// TwinCAT 3 PLC project PLC_Project
// ProgramVersion: 3.1.4026.19
// CompilerDefines: VISU_USEPROPERTYINFO,VISU_USEWSTRING
// libraries:
//   Tc2_Standard, * (Beckhoff Automation GmbH)
//   Tc2_System, * (Beckhoff Automation GmbH)
//   Tc2_Utilities, * (Beckhoff Automation GmbH)
//   Tc3_EventLogger, * (Beckhoff Automation GmbH)
//   VisuElemEventTable, * (System)
//   VisuSymbols, 4.5.0.0 (System)
// project tree:
//   DUTs/ ST_AlarmEventData_TextList.TcDUT, ST_AlarmEventData_Table.TcDUT
//   FBs/ FB_AlarmEx.TcPOU, FB_Message.TcPOU
//   / GlobalTextList.TcGTLO, PlcTask.TcTTO, Visualization Manager.TcVMO (not stored), VISU_TASK.TcTTO
//   GVLs/ HMI.TcGVL, SYS.TcGVL
//   POUs/ FB_AlarmLogEvent_TextList.TcPOU, FB_AlarmLogEvent_Table.TcPOU, MAIN.TcPOU
//   VISUs/ Alarms.TcVIS, Event_Table.TcVIS, Alarm_Table.TcVIS, Alarm_TextList.TcTLO, stAlarmEventData_TextList.TcTLO
//   VISUs/Frames/ AlarmRow.TcVIS, Alarm_Frame.TcVIS
// real-time tasks:
//   TASK PlcTask: cycle T#10ms, priority 20, ADS port 350
//   TASK VISU_TASK: cycle T#200000us, priority 30, ADS port 351
// I/O:
//   DEVICE Device 1 (EtherCAT) (disabled), AmsNetId 10.0.3.0.2.1
// variable links:
//   PLC_Project/PLC_Project Instance <-> Device 1 (EtherCAT)
//     PlcTask Inputs/MAIN.DevState <-> Inputs/DevState

CONFIGURATION PLC_Project
    RESOURCE PLC ON TwinCAT3
        TASK PlcTask(INTERVAL := T#10ms, PRIORITY := 20);
        TASK VISU_TASK(INTERVAL := T#200000us, PRIORITY := 30);
        PROGRAM MAIN WITH PlcTask : MAIN;
        PROGRAM VisuElems_Visu_Prg WITH VISU_TASK : VisuElems.Visu_Prg;
    END_RESOURCE
END_CONFIGURATION

// ---- DUTs/ST_AlarmEventData_TextList.TcDUT
TYPE ST_AlarmEventData_TextList :
STRUCT
	qActive		: BOOL;
	diEventID	: DINT;
	iClass		: INT; 		//0 = none, 1= Maintenance, 2= Message, 3= Hint, 4= StateInfo, 5= Instruction, 6 = Warning, 7= Alarm, 8= Parameter
	sTime		: STRING;
END_STRUCT
END_TYPE

// ---- DUTs/ST_AlarmEventData_Table.TcDUT
TYPE ST_AlarmEventData_Table :
STRUCT
	qActive		: BOOL;
	diEventID	: DINT;
	iClass		: INT; 		//0 = none, 1= Maintenance, 2= Message, 3= Hint, 4= StateInfo, 5= Instruction, 6 = Warning, 7= Alarm, 8= Parameter
	sTime		: STRING;
	sEvent		: STRING; 	// Event Text
END_STRUCT
END_TYPE

// ---- GVLs/HMI.TcGVL
{attribute 'qualified_only'}
VAR_GLOBAL
astActiveAlarmsList		: ARRAY [0..10] OF ST_AlarmEventData_TextList; // Display list of 10 active alarms, any more than that are just snowballs anyway so why display	
astActiveAlarmsTable	: ARRAY [1..50] OF ST_AlarmEventData_Table; // Display list of 50 active alarms
//Common Controls
	xFaultResetPB			: BOOL; //HMI Fault Reset PB
	xFaultPresent			: BOOL; //HMI Fault Present Indicator
END_VAR

// ---- GVLs/SYS.TcGVL
{attribute 'qualified_only'}
VAR_GLOBAL CONSTANT
iMaxSpeedConstant 		: INT := 60;
END_VAR

{attribute 'qualified_only'}
VAR_GLOBAL RETAIN
	
END_VAR

{attribute 'qualified_only'}
VAR_GLOBAL
	
//Program Declarations
	xFirstScan				: BOOL := TRUE;;
	xFaultPresent			: BOOL;
	ftrigFaultReset			: F_TRIG;
	xFaultReset				: BOOL;

//System Info
	fbGetLocalSystemTIme	: FB_LocalSystemTime;
	sSystemDateTime 		: STRING;
	sSystemTime 			: STRING;
	sSystemDate 			: STRING;
END_VAR

// ---- POUs/MAIN.TcPOU
PROGRAM MAIN
VAR
	DevState AT %I*			: UINT;
	fbReadEvents			: FB_ReadTc3Events; // Required for Event Table Visu Control
	fbMachineAlarm			: ARRAY[0..100] OF FB_AlarmEx;
	fbMachineMessage		: ARRAY[0..100] OF FB_Message;
	TestAlarm				: ARRAY[1..10] OF BOOL;
	TestMessage				: ARRAY[1..10] OF BOOL;
	
	ClearTable				: BOOL;
	VisuSeverity			: ARRAY[0..4] OF STRING := ['Verbose', 'Info', 'Warning', 'Error', 'Critical']; // Used in the Visu Combobox
	Severity				: TcEventSeverity;

	Fault 					: ARRAY [1..100] OF BOOL;
	fbAlarmLogEvent 		: ARRAY [1..100] OF FB_AlarmLogEvent_TextList; //Alarm Logging Event Handler
	fbAlarmLogEventTable	: ARRAY [1..100] OF FB_AlarmLogEvent_Table; //Alarm Logging Event Handler
	iFaultIndex				: INT;
	iAlarmClearIndex		: INT;
	iAlarmActiveIndex		: INT;
	iAlarmActiveIndex2		: INT;
	diAlarmEventLogIndex	: DINT;
END_VAR

//Get Local System Time
	SYS.fbGetLocalSystemTIme( 
		bEnable:= TRUE, 
		dwCycle:= 1);
	//Seperate Date and time
		SYS.sSystemDateTime := SYSTEMTIME_TO_STRING(in:= SYS.fbGetLocalSystemTIme.systemTime);
		SYS.sSystemDate := MID(STR:= SYS.sSystemDateTime, LEN:= 10 , POS:= 1 );
		SYS.sSystemTime := MID(STR:= SYS.sSystemDateTime, LEN:= 8 , POS:= 12 );

// HMI Fault PB Passthrough		
SYS.xFaultReset := HMI.xFaultResetPB;


	
// Twincat Event Logger	
// The function block enables the events of the TwinCAT 3 EventLogger to be displayed in the visualization element event table. 
// FB_ReadTc3Events is contained in the VisuElemEventTable library, which is automatically added to the project when the event table is activated
fbReadEvents(
	bReadEvents := TRUE,										// This input is used to enable the events to be read.
	nLanguageID := 1033,										// Defines which translation of the event text is to be retrieved. 1033 = English
	eDateAndTimeFormat := E_DateAndTimeFormat.en_US,			// Defines the format of the timestamps. E_DateAndTimeFormat
	bClearTable :=	ClearTable,					// The event table is cleared via a positive edge at this input. Alarms that were not acknowledged or reset are not removed from the table.
	eMinSeverity := Severity,									// Only events whose severity is at least as high as the severity specified here are displayed in the event table.
	aEvents => ,												// The function block uses this array to make the evaluated events available. The array can store a maximum of 80 messages. If the number of events is large, older messages are overwritten.
	nNumberOfEvents => ,										// Indicates how many events were triggered.
	bError => ,													// This output is set if an error occurs when polling or processing the events.
	hrErrorCode => );											// Indicates the error code of the error that has occurred.

Tc3_EventLogger();





// Legacy Alarm List
A99_Alarms_TextList();
A99_Alarms_Table();

// First Scan Complete
SYS.xFirstScan := FALSE;

ACTION A99_Alarms_Table:
//System Faults
	//Power Interrupted Fault							
		fbAlarmLogEventTable[1](
							i_diEventID:= 1,							// Must match the AlarmText Index for the message to display
							sEventText := 'Power Interrupt Fault',		// Enter an Event String Here
							i_iClassID:= 7,								// 0 = none, 1= Maintenance, 2= Message, 3= Hint, 4= StateInfo, 5= Instruction, 6 = Warning, 7= Alarm, 8= Paramater		
							bSetEvent := SYS.xFirstScan,				// Event activates on rising edge, clears on falling edge
							bLatchTillAck:= TRUE,						// Option to Latch alarm on even if no longer active, wait till alarm ack to clear
							bAck:= SYS.xFaultReset);					// Acknowledged and clears on rising edge if option LatchTillAck = false
							

		fbAlarmLogEventTable[2](
							i_diEventID:= 2,
							sEventText := 'Test Alarm 1',
							i_iClassID:= 7,
							bSetEvent := TestAlarm[1],
							bLatchTillAck:= TRUE,
							bAck:= SYS.xFaultReset);
							

		fbAlarmLogEventTable[3](
							i_diEventID:= 3,
							sEventText := 'Test Alarm 2',
							i_iClassID:= 2,
							bSetEvent := TestAlarm[2],
							bLatchTillAck:= TRUE,
							bAck:= SYS.xFaultReset);
							
					
		fbAlarmLogEventTable[4](
							i_diEventID:= 4,
							sEventText := 'Test Alarm 3',
							i_iClassID:= 6,
							bSetEvent := TestAlarm[3],
							bLatchTillAck:= TRUE,
							bAck:= SYS.xFaultReset);
							
				
		fbAlarmLogEventTable[5](
							i_diEventID:= 5,
							sEventText := 'Test Alarm 4',
							i_iClassID:= 7,
							bSetEvent := TestAlarm[4],
							bLatchTillAck:= TRUE,
							bAck:= SYS.xFaultReset);


// iClassID : 0 = none, 1= Maintenance, 2= Message, 3= Hint, 4= StateInfo, 5= Instruction, 6 = Warning, 7= Alarm, 8= Paramater	
//Monitor Fault Present
FOR iFaultIndex := 1 TO 100 BY 1 DO
	//System
	IF (iFaultIndex > 0) AND (iFaultIndex < 20) THEN // Look at Alarm Group 1-20
		IF fbAlarmLogEventTable[iFaultIndex].q_xActive AND (fbAlarmLogEventTable[iFaultIndex].i_iClassID = 7) THEN // Only Class 7 Count as Alarms
			SYS.xFaultPresent := TRUE;
		END_IF
	END_IF
	
(*  Some Other Alarm Group
	IF (iFaultIndex >= 20) AND (iFaultIndex < 40) THEN // Subsequent Alarm Group
		IF fbAlarmLogEvent[iFaultIndex].q_xActive AND (fbAlarmLogEvent[iFaultIndex].i_iClassID = 7) THEN
			OtherMachineFaultPreset := TRUE;
		END_IF
	END_IF
*)
END_FOR

// System Fault to HMI Fault Indicator
HMI.xFaultPresent := SYS.xFaultPresent;

IF SYS.xFaultReset THEN
	SYS.xFaultPresent := FALSE;
END_IF

(* Log all Alarms using the fbAlarmLogEvent function block*)
(* Alarm Text is in the Alarm_TextList File*)	

//Clear active alarms list before re-populating to ensure old cleared alarms are not stranded in the list
IF SYS.xFaultReset THEN
	FOR iAlarmClearIndex := 1 TO 50 BY 1 DO //10 possible active Alarms, no more!
		HMI.astActiveAlarmsTable[iAlarmClearIndex].sEvent := '';
		HMI.astActiveAlarmsTable[iAlarmClearIndex].diEventID := 0;
		HMI.astActiveAlarmsTable[iAlarmClearIndex].iClass := 0;
		HMI.astActiveAlarmsTable[iAlarmClearIndex].sTime := '';
	END_FOR;
END_IF
	
//Populate HMI Active Alarms list
	iAlarmActiveIndex2 := 0;  //Initialize before seeing how many active alarms there are.
	FOR diAlarmEventLogIndex := 1 TO 100 BY 1 DO //100 possible defined Alarms, no more!
		IF fbAlarmLogEvent[diAlarmEventLogIndex].q_xActive THEN
			IF iAlarmActiveIndex2 <= 9 THEN //10 max active alarms, no more!
				iAlarmActiveIndex2 := iAlarmActiveIndex2 + 1;
			END_IF
			HMI.astActiveAlarmsTable[iAlarmActiveIndex2].sEvent := fbAlarmLogEventTable[diAlarmEventLogIndex].q_stAlarmEventData.sEvent;
			HMI.astActiveAlarmsTable[iAlarmActiveIndex2].diEventID := fbAlarmLogEventTable[diAlarmEventLogIndex].q_stAlarmEventData.diEventID;
			HMI.astActiveAlarmsTable[iAlarmActiveIndex2].iClass := fbAlarmLogEventTable[diAlarmEventLogIndex].q_stAlarmEventData.iClass;
			IF HMI.astActiveAlarmsTable[iAlarmActiveIndex2].sTime = '' THEN
				HMI.astActiveAlarmsTable[iAlarmActiveIndex2].sTime := SYS.sSystemTime;
			END_IF
		END_IF
	END_FOR;
END_ACTION

ACTION A99_Alarms_TextList:
//System Faults
	//Power Interrupted Fault
		fbAlarmLogEvent[1](i_diEventID:= 1,					// Must match the AlarmText Index for the message to display
							i_iClassID:= 7,					// 0 = none, 1= Maintenance, 2= Message, 3= Hint, 4= StateInfo, 5= Instruction, 6 = Warning, 7= Alarm, 8= Paramater		
							bSetEvent := SYS.xFirstScan,	// Event activates on rising edge, clears on falling edge
							bLatchTillAck:= TRUE,			// Option to Latch alarm on even if no longer active, wait till alarm ack to clear
							bAck:= SYS.xFaultReset);		// Acknowledged and clears on rising edge if option LatchTillAck = false
							

		fbAlarmLogEvent[2](i_diEventID:= 2,
							i_iClassID:= 7,
							bSetEvent := TestAlarm[1],
							bLatchTillAck:= TRUE,
							bAck:= SYS.xFaultReset);
							

		fbAlarmLogEvent[3](i_diEventID:= 3,
							i_iClassID:= 2,
							bSetEvent := TestAlarm[2],
							bLatchTillAck:= TRUE,
							bAck:= SYS.xFaultReset);
							
					
		fbAlarmLogEvent[4](i_diEventID:= 4,
							i_iClassID:= 6,
							bSetEvent := TestAlarm[3],
							bLatchTillAck:= TRUE,
							bAck:= SYS.xFaultReset);
							
				
		fbAlarmLogEvent[5](i_diEventID:= 5,
							i_iClassID:= 7,
							bSetEvent := TestAlarm[4],
							bLatchTillAck:= TRUE,
							bAck:= SYS.xFaultReset);


// iClassID : 0 = none, 1= Maintenance, 2= Message, 3= Hint, 4= StateInfo, 5= Instruction, 6 = Warning, 7= Alarm, 8= Paramater	
//Monitor Fault Present
FOR iFaultIndex := 1 TO 100 BY 1 DO
	//System
	IF (iFaultIndex > 0) AND (iFaultIndex < 20) THEN // Look at Alarm Group 1-20
		IF fbAlarmLogEvent[iFaultIndex].q_xActive AND (fbAlarmLogEvent[iFaultIndex].i_iClassID = 7) THEN // Only Class 7 Count as Alarms
			SYS.xFaultPresent := TRUE;
		END_IF
	END_IF
	
(*  Some Other Alarm Group
	IF (iFaultIndex >= 20) AND (iFaultIndex < 40) THEN // Subsequent Alarm Group
		IF fbAlarmLogEvent[iFaultIndex].q_xActive AND (fbAlarmLogEvent[iFaultIndex].i_iClassID = 7) THEN
			OtherMachineFaultPreset := TRUE;
		END_IF
	END_IF
*)
END_FOR

// System Fault to HMI Fault Indicator
HMI.xFaultPresent := SYS.xFaultPresent;

IF SYS.xFaultReset THEN
	SYS.xFaultPresent := FALSE;
END_IF

(* Log all Alarms using the fbAlarmLogEvent function block*)
(* Alarm Text is in the Alarm_TextList File*)	

//Clear active alarms list before re-populating to ensure old cleared alarms are not stranded in the list
IF SYS.xFaultReset THEN
	FOR iAlarmClearIndex := 0 TO 10 BY 1 DO //10 possible active Alarms, no more!
		HMI.astActiveAlarmsList[iAlarmClearIndex].diEventID := 0;
		HMI.astActiveAlarmsList[iAlarmClearIndex].iClass := 0;
		HMI.astActiveAlarmsList[iAlarmClearIndex].sTime := '';
	END_FOR;
END_IF
	
//Populate HMI Active Alarms list
	iAlarmActiveIndex := 0;  //Initialize before seeing how many active alarms there are.
	FOR diAlarmEventLogIndex := 1 TO 100 BY 1 DO //100 possible defined Alarms, no more!
		IF fbAlarmLogEvent[diAlarmEventLogIndex].q_xActive THEN
			IF iAlarmActiveIndex <= 9 THEN //10 max active alarms, no more!
				iAlarmActiveIndex := iAlarmActiveIndex + 1;
			END_IF
			HMI.astActiveAlarmsList[iAlarmActiveIndex].diEventID := fbAlarmLogEvent[diAlarmEventLogIndex].q_stAlarmEventData.diEventID;
			HMI.astActiveAlarmsList[iAlarmActiveIndex].iClass := fbAlarmLogEvent[diAlarmEventLogIndex].q_stAlarmEventData.iClass;
			IF HMI.astActiveAlarmsList[iAlarmActiveIndex].sTime = '' THEN
				HMI.astActiveAlarmsList[iAlarmActiveIndex].sTime := SYS.sSystemTime;
			END_IF
		END_IF
	END_FOR;
END_ACTION

ACTION TC3_EventLogger:
// Event Classes are created in System -> Type System -> Event Class
// Write Click and Create your new Event Class.

fbMachineMessage[1](
	evtEntry:= TC_EVENTS.Test_EventClass.Test_Message1, 
	bEvt:= TestMessage[1]);
	
fbMachineMessage[2](
	evtEntry:= TC_EVENTS.Test_EventClass.Test_Message2, 
	bEvt:= TestMessage[2]);
	
fbMachineMessage[3](
	evtEntry:= TC_EVENTS.Test_EventClass.Test_Message3, 
	bEvt:= TestMessage[3]);
	
fbMachineMessage[4](
	evtEntry:= TC_EVENTS.Test_EventClass.Test_Message4, 
	bEvt:= TestMessage[4]);
	
fbMachineMessage[5](
	evtEntry:= TC_EVENTS.Test_EventClass.Test_Message5, 
	bEvt:= TestMessage[5]);
	
fbMachineAlarm[1](
	evtEntry:= TC_EVENTS.Test_EventClass.PowerInterrupt, 
	bEvt:= SYS.xFirstScan,
	bConfirm := SYS.xFaultReset); 
	
fbMachineAlarm[2](
	evtEntry:= TC_EVENTS.Test_EventClass.Test_Event1, 
	bEvt:= TestAlarm[1],
	bConfirm := SYS.xFaultReset); 
	
fbMachineAlarm[3](
	evtEntry:= TC_EVENTS.Test_EventClass.Test_Event2, 
	bEvt:= TestAlarm[2],
	bConfirm := SYS.xFaultReset); 
	
fbMachineAlarm[4](
	evtEntry:= TC_EVENTS.Test_EventClass.Test_Event3, 
	bEvt:= TestAlarm[3],
	bConfirm := SYS.xFaultReset); 
	
fbMachineAlarm[5](
	evtEntry:= TC_EVENTS.Test_EventClass.Test_Event4, 
	bEvt:= TestAlarm[4],
	bConfirm := SYS.xFaultReset); 


// Trigger Several Alarms At Once below.
// Change Severity in the Event Class	
	
fbMachineAlarm[6](
	evtEntry:= TC_EVENTS.Events._IECCONF_1, 
	bEvt:= TestAlarm[5],
	bConfirm := SYS.xFaultReset); 
	
fbMachineAlarm[7](
	evtEntry:= TC_EVENTS.Events._IECCONF_2, 
	bEvt:= TestAlarm[5],
	bConfirm := SYS.xFaultReset);
	
fbMachineAlarm[8](
	evtEntry:= TC_EVENTS.Events._IECCONF_3, 
	bEvt:= TestAlarm[5],
	bConfirm := SYS.xFaultReset);
	
fbMachineAlarm[9](
	evtEntry:= TC_EVENTS.Events._IECCONF_4, 
	bEvt:= TestAlarm[5],
	bConfirm := SYS.xFaultReset);
	
fbMachineAlarm[10](
	evtEntry:= TC_EVENTS.Events._IECCONF_5, 
	bEvt:= TestAlarm[5],
	bConfirm := SYS.xFaultReset);
	
fbMachineAlarm[11](
	evtEntry:= TC_EVENTS.Events._IECCONF_6, 
	bEvt:= TestAlarm[5],
	bConfirm := SYS.xFaultReset);
	
fbMachineAlarm[12](
	evtEntry:= TC_EVENTS.Events._IECCONF_7, 
	bEvt:= TestAlarm[5],
	bConfirm := SYS.xFaultReset);
	
fbMachineAlarm[13](
	evtEntry:= TC_EVENTS.Events._IECCONF_8, 
	bEvt:= TestAlarm[5],
	bConfirm := SYS.xFaultReset);
	
fbMachineAlarm[14](
	evtEntry:= TC_EVENTS.Events._IECCONF_9, 
	bEvt:= TestAlarm[5],
	bConfirm := SYS.xFaultReset);
	
fbMachineAlarm[15](
	evtEntry:= TC_EVENTS.Events._IECCONF_10, 
	bEvt:= TestAlarm[5],
	bConfirm := SYS.xFaultReset);
	
fbMachineAlarm[16](
	evtEntry:= TC_EVENTS.Events._IECCONF_11, 
	bEvt:= TestAlarm[5],
	bConfirm := SYS.xFaultReset);
	
fbMachineAlarm[17](
	evtEntry:= TC_EVENTS.Events._IECCONF_12, 
	bEvt:= TestAlarm[5],
	bConfirm := SYS.xFaultReset);
	
fbMachineAlarm[18](
	evtEntry:= TC_EVENTS.Events._IECCONF_13, 
	bEvt:= TestAlarm[5],
	bConfirm := SYS.xFaultReset);
	
fbMachineAlarm[19](
	evtEntry:= TC_EVENTS.Events._IECCONF_14, 
	bEvt:= TestAlarm[5],
	bConfirm := SYS.xFaultReset);
	
fbMachineAlarm[20](
	evtEntry:= TC_EVENTS.Events._IECCONF_15, 
	bEvt:= TestAlarm[5],
	bConfirm := SYS.xFaultReset);
	
fbMachineAlarm[21](
	evtEntry:= TC_EVENTS.Events._IECCONF_16, 
	bEvt:= TestAlarm[5],
	bConfirm := SYS.xFaultReset);
	
fbMachineAlarm[22](
	evtEntry:= TC_EVENTS.Events._IECCONF_17, 
	bEvt:= TestAlarm[5],
	bConfirm := SYS.xFaultReset);
END_ACTION

END_PROGRAM

// ---- FBs/FB_AlarmEx.TcPOU
FUNCTION_BLOCK FB_AlarmEx EXTENDS FB_TcAlarm
VAR_INPUT
	evtEntry	: TcEventEntry;
	bEvt		: BOOL;
	bConfirm	: BOOL;
END_VAR
VAR_OUTPUT
END_VAR
VAR
	SourceInfo	: FB_TcSourceInfo;
	bInit	: BOOL := TRUE;
	bMem	: BOOL;
END_VAR

IF bInit THEN
	SUPER^.CreateEx(evtEntry, (evtentry.eSeverity = TcEventSeverity.Critical) OR (evtentry.eSeverity = TcEventSeverity.Error), 0);
	bInit := FALSE;
END_IF

IF bEvt AND NOT bMem AND SUPER^.eConfirmationState <> TcEventConfirmationState.WaitForConfirmation THEN
	SUPER^.Raise(0);
END_IF

IF bMem AND NOT bEvt THEN
	SUPER^.Clear(0,FALSE);
END_IF

IF bConfirm THEN
	SUPER^.Confirm(0);
END_IF

bMem := bEvt;

END_FUNCTION_BLOCK

// ---- FBs/FB_Message.TcPOU
FUNCTION_BLOCK FB_Message EXTENDS FB_TcMessage
VAR_INPUT
	evtEntry	: TcEventEntry;
	bEvt		: BOOL;
END_VAR
VAR_OUTPUT
	bSent		: BOOL;
END_VAR
VAR
	rtrigSend	: R_TRIG;
	bInit	: BOOL := TRUE;
	bMem	: BOOL;
END_VAR

bSent := FALSE;
IF bInit THEN
	SUPER^.CreateEx(stEventEntry := evtEntry, ipSourceInfo := 0);
	bInit := FALSE;
END_IF

rtrigSend(CLK:= bEvt);
IF rtrigSend.Q THEN
	SUPER^.Send(0);
	bSent := TRUE;
END_IF

END_FUNCTION_BLOCK

// ---- POUs/FB_AlarmLogEvent_TextList.TcPOU
FUNCTION_BLOCK FB_AlarmLogEvent_TextList
VAR_INPUT
	bSetEvent			: BOOL;	//Trigger to activate the Alarm
	i_diEventID			: DINT;
	i_iClassID			: INT;
	bLatchTillAck 		: BOOL; //Latch Alarm active till Acked even if alarm event clears.
	bAck				: BOOL; //Acknowledge the alarm and clear it.
	tsTime				:TIMESTRUCT;
END_VAR
VAR_OUTPUT
	q_stAlarmEventData	: ST_AlarmEventData_TextList;
	q_xActive			: BOOL;
END_VAR
VAR
	fbFormatString		: FB_FormatString;
END_VAR

//Why use a Function Block?
//So we could add a active time/date stamp
//So we could add to a historical alarm area
//So we could add ack requirment if decided one was needed.

//Monitor when Alarm is active, save data
	IF bSetEvent AND NOT q_xActive THEN 
		q_xActive	:= TRUE;
		q_stAlarmEventData.diEventID := i_diEventID;
		q_stAlarmEventData.iClass := i_iClassID;
		fbFormatString(sFormat := '%d:%d:%d',
						arg1 := F_word(tsTime.wHour),
						arg2 := F_word(tsTime.wMinute),
						arg3 := F_word(tsTime.wSecond),
						sOut => q_stAlarmEventData.sTime );	
	ELSIF NOT bSetEvent AND NOT bLatchTillAck THEN
		q_xActive := FALSE;
	END_IF;

//Alarm no longer active
	IF bLatchTillAck AND q_xActive AND bAck THEN
		q_xActive := FALSE;
	END_IF

END_FUNCTION_BLOCK

// ---- POUs/FB_AlarmLogEvent_Table.TcPOU
FUNCTION_BLOCK FB_AlarmLogEvent_Table
VAR_INPUT
	bSetEvent			: BOOL;	//Trigger to activate the Alarm
	sEventText			: STRING;
	i_diEventID			: DINT;
	i_iClassID			: INT;
	bLatchTillAck 		: BOOL; //Latch Alarm active till Acked even if alarm event clears.
	bAck				: BOOL; //Acknowledge the alarm and clear it.
	tsTime				:TIMESTRUCT;
END_VAR
VAR_OUTPUT
	q_stAlarmEventData	: ST_AlarmEventData_Table;
	q_xActive			: BOOL;
END_VAR
VAR
	fbFormatString		: FB_FormatString;
END_VAR

//Why use a Function Block?
//So we could add a active time/date stamp
//So we could add to a historical alarm area
//So we could add ack requirment if decided one was needed.

//Monitor when Alarm is active, save data
	IF bSetEvent AND NOT q_xActive THEN 
		q_xActive	:= TRUE;
		q_stAlarmEventData.sEvent := sEventText;
		q_stAlarmEventData.diEventID := i_diEventID;
		q_stAlarmEventData.iClass := i_iClassID;
		fbFormatString(sFormat := '%d:%d:%d',
						arg1 := F_word(tsTime.wHour),
						arg2 := F_word(tsTime.wMinute),
						arg3 := F_word(tsTime.wSecond),
						sOut => q_stAlarmEventData.sTime );	
	ELSIF NOT bSetEvent AND NOT bLatchTillAck THEN
		q_xActive := FALSE;
	END_IF;

//Alarm no longer active
	IF bLatchTillAck AND q_xActive AND bAck THEN
		q_xActive := FALSE;
	END_IF

END_FUNCTION_BLOCK

// ---- GlobalTextList.TcGTLO
TEXTLIST GlobalTextList
  481 = ' ** Table Displays 80 Alarms, and Overwrites the Oldest'
  566 = ' ** The Event Table Displays 80 Alarms, and Overwrites the Oldest'
  60 = ' ** The Event Table displays 80 Alarms, and overwrites the oldest'
  900 = '%s'
  882 = '* This Filters incoming Alarms, not currently displayed Alarms.'
  21 = '* This Severity Filters incoming Alarms, not currently displayed Alarms.'
  243 = '*** Only events whose severity is at least as high as the severity specified here are displayed in the event table.'
  652 = '*** Only events whose severity is at least as high as the severity specified here are displayed in the event table.  This does not effect currently displayed events, only incoming.'
  807 = 'Active'
  504 = 'Alarm List Utilizing Frames and Text List This utilized FB_AlarmLogEvent_TextList'
  73 = 'Alarm Table '
  909 = 'Alarm Table Utilizing Frames and Text List'
  872 = 'Alarm Table Utilizing Frames and Text List This utilized FB_AlarmLogEvent_TextList'
  335 = 'Alarm Table Utilizing Frames and Text List \\n Utilize'
  947 = 'Back'
  153 = 'Class'
  653 = 'CLASS'
  568 = 'Clear'
  27 = 'Clear Table'
  497 = 'EVENT'
  360 = 'Event ID'
  151 = 'Event Logger'
  480 = 'Event Table'
  578 = 'Event Table - This is the recommended control'
  837 = 'Event Table - This is the recommended control.'
  738 = 'Event Table - This is the recommended control.  Table Displays 80 Alarms, and Overwrites the Oldest'
  994 = 'Frame Example'
  126 = 'HMI.astActiveAlarmsTable[INDEX].qActive'
  487 = 'id'
  871 = 'ID'
  140 = 'Only events whose severity is at least as high as the severity specified here are displayed in the event table.'
  707 = 'Reset'
  37 = 'Table Example'
  458 = 'Time'
  376 = 'TIME'
END_TEXTLIST

// ---- VISUs/Alarms.TcVIS
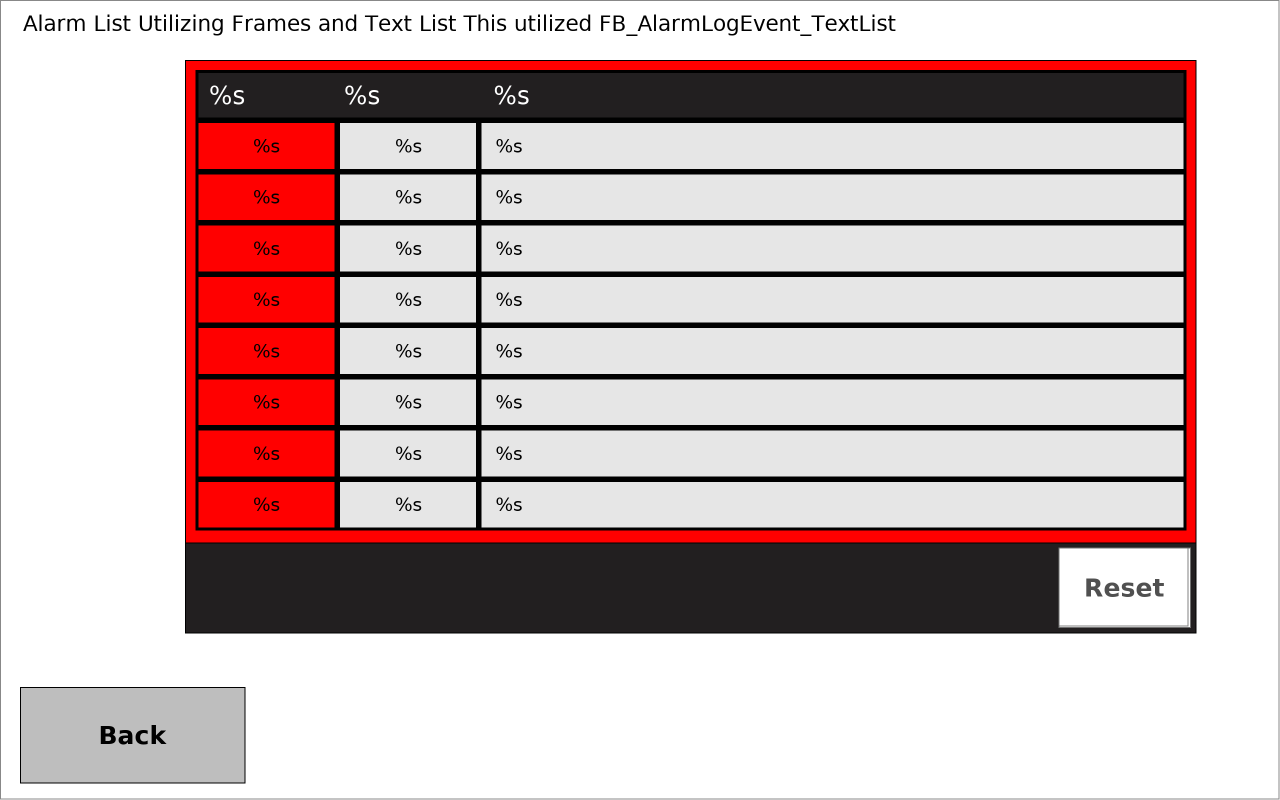
VISUALIZATION Alarms  // 1280x800
    Rectangle (20,9 909x60), "Alarm List Utilizing Frames and Text List This utilized FB_AlarmLogEvent_TextList"
    Frame (185,60 1011x573)
        shows Alarm_Frame(xFaultResetPB := HMI.xFaultResetPB, sAlarmTextList := 'Alarm_TextList', sEventDataTextList := 'stAlarmEventData_TextList', astActiveAlarmsList_1 := HMI.astActiveAlarmsList[1], astActiveAlarmsList_2 := HMI.astActiveAlarmsList[2], astActiveAlarmsList_3 := HMI.astActiveAlarmsList[3], astActiveAlarmsList_4 := HMI.astActiveAlarmsList[4], astActiveAlarmsList_5 := HMI.astActiveAlarmsList[5], astActiveAlarmsList_6 := HMI.astActiveAlarmsList[6], astActiveAlarmsList_7 := HMI.astActiveAlarmsList[7], astActiveAlarmsList_8 := HMI.astActiveAlarmsList[8])
    Rectangle (20,687 225x96), "Back"
        OnMouseClick: change screen: Previous Alarm_Table
END_VISUALIZATION

// ---- VISUs/Event_Table.TcVIS
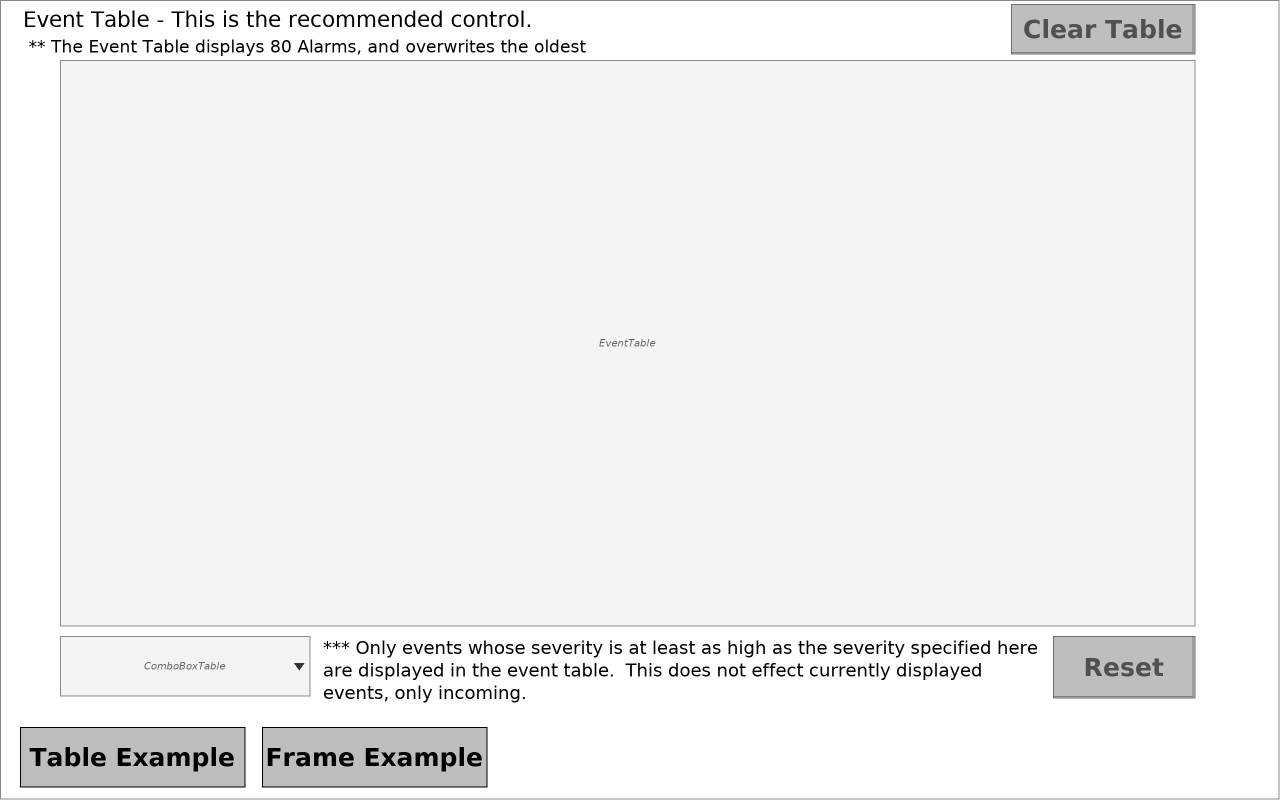
VISUALIZATION Event_Table  // 1280x800
    Rectangle (20,5 909x30), "Event Table - This is the recommended control."
    Rectangle (20,727 225x60), "Table Example"
        OnMouseClick: change screen: Alarm_Table
    Button (1053,636 142x62), "Reset"
        tap HMI.xFaultResetPB
    Rectangle (262,727 225x60), "Frame Example"
        OnMouseClick: change screen: Alarms
    ComboBoxTable (60,636 250x60), variable: MAIN.Severity, data array: MAIN.VisuSeverity
        p1014161805: 4 - 0 + INT#1
        p3854506369: MAIN.VisuSeverity[INDEX]
    Button (1011,4 184x50), "Clear Table"
        tap MAIN.ClearTable
    Rectangle (20,35 909x30), "** The Event Table displays 80 Alarms, and overwrites the oldest"
    EventTable (60,60 1135x566)
        p1690906150: Class
        p3258520714: Date
        p2231227367: Time
        p3993844394: Event
        p2076579579: Details
        p3558512729: MAIN.fbReadEvents.aEvents
        p3921149237: m_pDataArray..pArray
    Label (320,626 734x89), "*** Only events whose severity is at least as high as the severity specified here are displayed in the event table. This does not effect currently displayed events, only incoming."
END_VISUALIZATION

// ---- VISUs/Alarm_Table.TcVIS
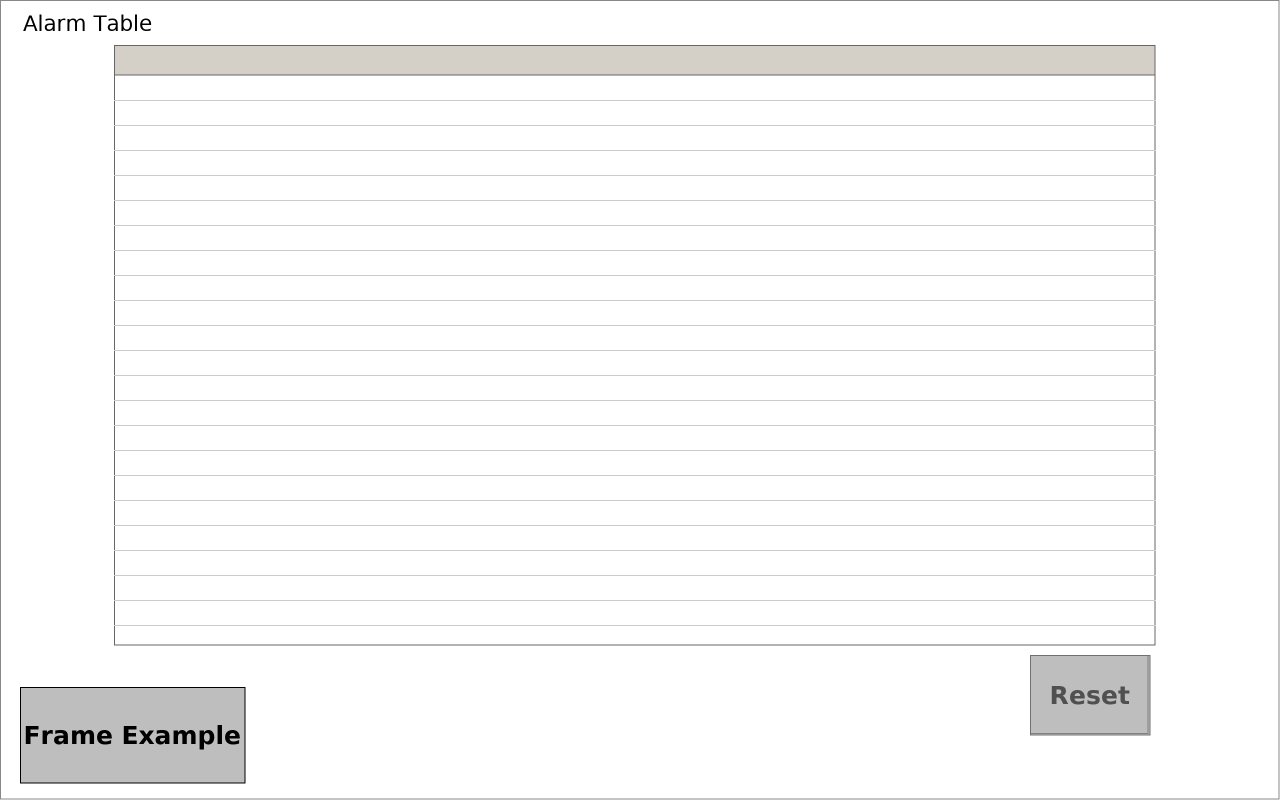
VISUALIZATION Alarm_Table  // 1280x800
    Rectangle (20,9 909x60), "Alarm Table"
    Table (114,45 1041x600), text list: 'Alarm_TextList', data array: HMI.astActiveAlarmsTable
        p1014161805: 50 - 1 + INT#1
        p3854506369: HMI.astActiveAlarmsTable[INDEX].qActive
        p1892666644: HMI.astActiveAlarmsTable[INDEX].diEventID
        p338671338: HMI.astActiveAlarmsTable[INDEX].iClass
        p2170511999: HMI.astActiveAlarmsTable[INDEX].sTime
        p3723444502: HMI.astActiveAlarmsTable[INDEX].sEvent
    Rectangle (20,687 225x96), "Frame Example"
        OnMouseClick: change screen: Alarms
    Button (1030,655 120x80), "Reset"
        tap HMI.xFaultResetPB
END_VISUALIZATION

// ---- VISUs/Alarm_TextList.TcTLO
TEXTLIST Alarm_TextList
  1 = 'Power Interrupted Fault'
  2 = 'Test 1'
  3 = 'Test 2'
  4 = 'Test 3'
  5 = 'Test 4'
   = ''
END_TEXTLIST

// ---- VISUs/Frames/AlarmRow.TcVIS
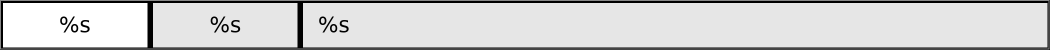
VISUALIZATION AlarmRow  // 1050x50
VAR_IN_OUT

	
END_VAR

VAR_INPUT
	sAlarmTextList 	: STRING;
	sEventDataTextList : STRING;
	stAlarmLogEvent : ST_AlarmEventData_TextList;
END_VAR
    Rectangle (0,0 150x50), "%s", text variable: stAlarmLogEvent.sTime, colour toggle: stAlarmLogEvent.iClass = 7
    Rectangle (300,0 750x50), colour toggle: stAlarmLogEvent.iClass = 7, text list: ''
    Rectangle (150,0 150x50), colour toggle: stAlarmLogEvent.iClass = 7, text list: ''
    Textfield (315,10 721x30), "%s", invisible if: stAlarmLogEvent.diEventID = 0, text list: sAlarmTextList, text index: stAlarmLogEvent.diEventID
    Textfield (159,10 133x30), "%s", invisible if: stAlarmLogEvent.diEventID = 0, text list: sEventDataTextList, text index: stAlarmLogEvent.iClass
END_VISUALIZATION

// ---- VISUs/Frames/Alarm_Frame.TcVIS
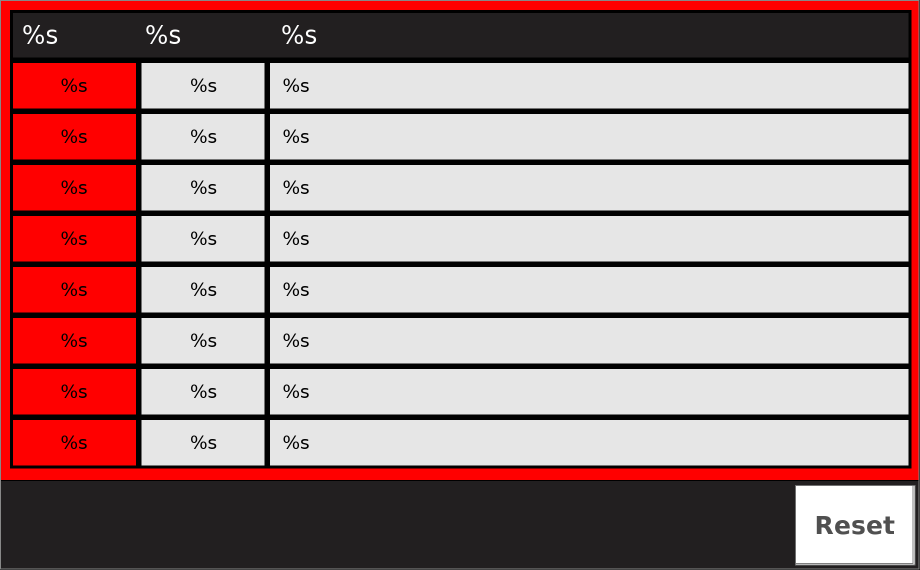
VISUALIZATION Alarm_Frame  // 920x570
VAR_IN_OUT
	xFaultResetPB : BOOL;
END_VAR

VAR_INPUT
	sAlarmTextList 	: STRING;
	sEventDataTextList : STRING;
	astActiveAlarmsList_1 : ST_AlarmEventData_TextList;
	astActiveAlarmsList_2 : ST_AlarmEventData_TextList;
	astActiveAlarmsList_3 : ST_AlarmEventData_TextList;
	astActiveAlarmsList_4 : ST_AlarmEventData_TextList;
	astActiveAlarmsList_5 : ST_AlarmEventData_TextList;
	astActiveAlarmsList_6 : ST_AlarmEventData_TextList;
	astActiveAlarmsList_7 : ST_AlarmEventData_TextList;
	astActiveAlarmsList_8 : ST_AlarmEventData_TextList;
END_VAR

VAR_OUTPUT
	
END_VAR
    Rectangle (0,0 920x570)
    Frame (10,60 901x51)
        shows AlarmRow(sAlarmTextList := sAlarmTextList, sEventDataTextList := sEventDataTextList, stAlarmLogEvent := astActiveAlarmsList_1)
    Frame (10,111 901x51)
        shows AlarmRow(sAlarmTextList := sAlarmTextList, sEventDataTextList := sEventDataTextList, stAlarmLogEvent := astActiveAlarmsList_2)
    Frame (10,213 901x51)
        shows AlarmRow(sAlarmTextList := sAlarmTextList, sEventDataTextList := sEventDataTextList, stAlarmLogEvent := astActiveAlarmsList_4)
    Frame (10,162 901x51)
        shows AlarmRow(sAlarmTextList := sAlarmTextList, sEventDataTextList := sEventDataTextList, stAlarmLogEvent := astActiveAlarmsList_3)
    Frame (10,264 901x51)
        shows AlarmRow(sAlarmTextList := sAlarmTextList, sEventDataTextList := sEventDataTextList, stAlarmLogEvent := astActiveAlarmsList_5)
    Frame (10,315 901x51)
        shows AlarmRow(sAlarmTextList := sAlarmTextList, sEventDataTextList := sEventDataTextList, stAlarmLogEvent := astActiveAlarmsList_6)
    Frame (10,366 901x51)
        shows AlarmRow(sAlarmTextList := sAlarmTextList, sEventDataTextList := sEventDataTextList, stAlarmLogEvent := astActiveAlarmsList_7)
    Frame (10,417 901x51)
        shows AlarmRow(sAlarmTextList := sAlarmTextList, sEventDataTextList := sEventDataTextList)
    Rectangle (10,10 901x50)
    Textfield (19,15 120x40), "%s", text list: sAlarmTextList, text index: 101
    Textfield (278,15 628x40), "%s", text list: sAlarmTextList, text index: 102
    Rectangle (0,480 920x90)
    Textfield (142,15 120x40), "%s", text list: sAlarmTextList, text index: 103
    Button (795,485 120x80), "Reset"
        tap xFaultResetPB
END_VISUALIZATION

// ---- VISUs/stAlarmEventData_TextList.TcTLO
TEXTLIST stAlarmEventData_TextList
  0 = ''
  1 = 'Maintenance'
  2 = 'Message'
  3 = 'Hint'
  4 = 'StateInfo'
  5 = 'Instruction'
  6 = 'Warning'
  7 = 'Alarm'
  8 = 'Parameter'
   = ''
END_TEXTLIST
